# EPICS autosave request: iocs/eigerIOC/iocBoot/iocPilatus4/auto_settings.req
file "eiger2_settings.req",       P=$(P),  R=cam1:
file "NDStdArrays_settings.req",  P=$(P),  R=image1:
file "NDStdArrays_settings.req",  P=$(P),  R=image2:
file "commonPlugin_settings.req", P=$(P)
